// TIA Portal V19 export
VAR_GLOBAL   // PLC tag table "Equipment_Template_DefaultTagTable_11"
   "Tag_49(7)" AT %I30042.0 : Bool;   // 物流线允许出
   "Tag_50(7)" AT %I30042.1 : Bool;   // 物流线通知托盘送出完成
   "Tag_51(7)" AT %I30042.2 : Bool;   // 物流线收到单机收到的物流线出到位信号
   "Tag_52(7)" AT %I30042.3 : Bool;   // 物流线空闲
   "Tag_53(7)" AT %I30042.4 : Bool;
   "Tag_54(7)" AT %I30042.5 : Bool;
   "Tag_55(7)" AT %I30042.6 : Bool;
   "Tag_56(7)" AT %I30042.7 : Bool;   // 物流请求出托盘
   "Tag_57(7)" AT %I30043.0 : Bool;   // 物流线忙碌
   "Tag_58(7)" AT %I30043.1 : Bool;   // 物流线收到单机返回出到位信号
   "Tag_59(7)" AT %I30043.2 : Bool;   // 物流工位报警
   "Tag_60(7)" AT %I30043.3 : Bool;   // 物流有拖盘待出
   "Tag_61(7)" AT %I30043.4 : Bool;
   "Tag_62(7)" AT %I30043.5 : Bool;
   "Tag_63(7)" AT %I30043.6 : Bool;
   "Tag_64(7)" AT %I30043.7 : Bool;
END_VAR
